Staubli VAL3: Prefix.pjx

--- Prefix.pjx ---
Parameters version=s7.7.2 stackSize=5000 millimeterUnit=true
Program file=start.pgx
Program file=stop.pgx
Data file=Prefix.dtx

--- Prefix.dtx ---
mdesc mNomSpeed
public num nLength
